TYPE U_Syntax_Union : UNION
        dwRaw  : DWORD;
        fValue : REAL;
        aBytes : ARRAY[0..3] OF BYTE;
        nInt32 : DINT;
    END_UNION
END_TYPE

(* stored: Version 1.1.0.1, ProductVersion 3.1.4024.16
   DUT U_Syntax_Union: Id {bd1ef978-742e-44fd-8696-5e9fa8e2bfa7} *)
